(* CoDeSys 2.3.9.52 project: dom1.pro *)
(* Libraries: Standard.lib 8.11.10 11:37:48, SYSLIBCALLBACK.LIB 8.11.10 11:37:48 *)

(* PLC configuration (modules and I/O channels)
0750-0430 8 DI 24 V DC 3.0ms [Type_1_8_Channels] node 0, in %IB0 out %QB0 {INTTypePAAssignment = PLC; INTTypeModule = plugged}
  AT %IX0.0 [BOOLOnX_I] Ch_1 Digital input
  AT %IX0.1 [BOOLOnX_I] Ch_2 Digital input
  AT %IX0.2 [BOOLOnX_I] Ch_3 Digital input
  AT %IX0.3 [BOOLOnX_I] Ch_4 Digital input
  AT %IX0.4 [BOOLOnX_I] Ch_5 Digital input
  AT %IX0.5 [BOOLOnX_I] Ch_6 Digital input
  AT %IX0.6 [BOOLOnX_I] Ch_7 Digital input
  AT %IX0.7 [BOOLOnX_I] Ch_8 Digital input
0750-0430 8 DI 24 V DC 3.0ms [Type_1_8_Channels] node 1, in %IB0 out %QB0 {INTTypePAAssignment = PLC; INTTypeModule = plugged}
  AT %IX0.8 [BOOLOnX_I] Ch_1 Digital input
  AT %IX0.9 [BOOLOnX_I] Ch_2 Digital input
  AT %IX0.10 [BOOLOnX_I] Ch_3 Digital input
  AT %IX0.11 [BOOLOnX_I] Ch_4 Digital input
  AT %IX0.12 [BOOLOnX_I] Ch_5 Digital input
  AT %IX0.13 [BOOLOnX_I] Ch_6 Digital input
  AT %IX0.14 [BOOLOnX_I] Ch_7 Digital input
  AT %IX0.15 [BOOLOnX_I] Ch_8 Digital input
0750-0430 8 DI 24 V DC 3.0ms [Type_1_8_Channels] node 2, in %IB1 out %QB0 {INTTypePAAssignment = PLC; INTTypeModule = plugged}
  AT %IX1.0 [BOOLOnX_I] Ch_1 Digital input
  AT %IX1.1 [BOOLOnX_I] Ch_2 Digital input
  AT %IX1.2 [BOOLOnX_I] Ch_3 Digital input
  AT %IX1.3 [BOOLOnX_I] Ch_4 Digital input
  AT %IX1.4 [BOOLOnX_I] Ch_5 Digital input
  AT %IX1.5 [BOOLOnX_I] Ch_6 Digital input
  AT %IX1.6 [BOOLOnX_I] Ch_7 Digital input
  AT %IX1.7 [BOOLOnX_I] Ch_8 Digital input
0750-0430 8 DI 24 V DC 3.0ms [Type_1_8_Channels] node 3, in %IB2 out %QB0 {INTTypePAAssignment = PLC; INTTypeModule = plugged}
  AT %IX1.8 [BOOLOnX_I] Ch_1 Digital input
  AT %IX1.9 [BOOLOnX_I] Ch_2 Digital input
  AT %IX1.10 [BOOLOnX_I] Ch_3 Digital input
  AT %IX1.11 [BOOLOnX_I] Ch_4 Digital input
  AT %IX1.12 [BOOLOnX_I] Ch_5 Digital input
  AT %IX1.13 [BOOLOnX_I] Ch_6 Digital input
  AT %IX1.14 [BOOLOnX_I] Ch_7 Digital input
  AT %IX1.15 [BOOLOnX_I] Ch_8 Digital input
0750-0430 8 DI 24 V DC 3.0ms [Type_1_8_Channels] node 4, in %IB3 out %QB0 {INTTypePAAssignment = PLC; INTTypeModule = plugged}
  AT %IX2.0 [BOOLOnX_I] Ch_1 Digital input
  AT %IX2.1 [BOOLOnX_I] Ch_2 Digital input
  AT %IX2.2 [BOOLOnX_I] Ch_3 Digital input
  AT %IX2.3 [BOOLOnX_I] Ch_4 Digital input
  AT %IX2.4 [BOOLOnX_I] Ch_5 Digital input
  AT %IX2.5 [BOOLOnX_I] Ch_6 Digital input
  AT %IX2.6 [BOOLOnX_I] Ch_7 Digital input
  AT %IX2.7 [BOOLOnX_I] Ch_8 Digital input
0750-0430 8 DI 24 V DC 3.0ms [Type_1_8_Channels] node 5, in %IB4 out %QB0 {INTTypePAAssignment = PLC; INTTypeModule = plugged}
  AT %IX2.8 [BOOLOnX_I] Ch_1 Digital input
  AT %IX2.9 [BOOLOnX_I] Ch_2 Digital input
  AT %IX2.10 [BOOLOnX_I] Ch_3 Digital input
  AT %IX2.11 [BOOLOnX_I] Ch_4 Digital input
  AT %IX2.12 [BOOLOnX_I] Ch_5 Digital input
  AT %IX2.13 [BOOLOnX_I] Ch_6 Digital input
  AT %IX2.14 [BOOLOnX_I] Ch_7 Digital input
  AT %IX2.15 [BOOLOnX_I] Ch_8 Digital input
0750-0430 8 DI 24 V DC 3.0ms [Type_1_8_Channels] node 6, in %IB5 out %QB0 {INTTypePAAssignment = PLC; INTTypeModule = plugged}
  AT %IX3.0 [BOOLOnX_I] Ch_1 Digital input
  AT %IX3.1 [BOOLOnX_I] Ch_2 Digital input
  AT %IX3.2 [BOOLOnX_I] Ch_3 Digital input
  AT %IX3.3 [BOOLOnX_I] Ch_4 Digital input
  AT %IX3.4 [BOOLOnX_I] Ch_5 Digital input
  AT %IX3.5 [BOOLOnX_I] Ch_6 Digital input
  AT %IX3.6 [BOOLOnX_I] Ch_7 Digital input
  AT %IX3.7 [BOOLOnX_I] Ch_8 Digital input
0750-0430 8 DI 24 V DC 3.0ms [Type_1_8_Channels] node 7, in %IB6 out %QB0 {INTTypePAAssignment = PLC; INTTypeModule = plugged}
  AT %IX3.8 [BOOLOnX_I] Ch_1 Digital input
  AT %IX3.9 [BOOLOnX_I] Ch_2 Digital input
  AT %IX3.10 [BOOLOnX_I] Ch_3 Digital input
  AT %IX3.11 [BOOLOnX_I] Ch_4 Digital input
  AT %IX3.12 [BOOLOnX_I] Ch_5 Digital input
  AT %IX3.13 [BOOLOnX_I] Ch_6 Digital input
  AT %IX3.14 [BOOLOnX_I] Ch_7 Digital input
  AT %IX3.15 [BOOLOnX_I] Ch_8 Digital input
0750-0430 8 DI 24 V DC 3.0ms [Type_1_8_Channels] node 8, in %IB7 out %QB0 {INTTypePAAssignment = PLC; INTTypeModule = plugged}
  AT %IX4.0 [BOOLOnX_I] Ch_1 Digital input
  AT %IX4.1 [BOOLOnX_I] Ch_2 Digital input
  AT %IX4.2 [BOOLOnX_I] Ch_3 Digital input
  AT %IX4.3 [BOOLOnX_I] Ch_4 Digital input
  AT %IX4.4 [BOOLOnX_I] Ch_5 Digital input
  AT %IX4.5 [BOOLOnX_I] Ch_6 Digital input
  AT %IX4.6 [BOOLOnX_I] Ch_7 Digital input
  AT %IX4.7 [BOOLOnX_I] Ch_8 Digital input
0750-0430 8 DI 24 V DC 3.0ms [Type_1_8_Channels] node 9, in %IB8 out %QB0 {INTTypePAAssignment = PLC; INTTypeModule = plugged}
  AT %IX4.8 [BOOLOnX_I] Ch_1 Digital input
  AT %IX4.9 [BOOLOnX_I] Ch_2 Digital input
  AT %IX4.10 [BOOLOnX_I] Ch_3 Digital input
  AT %IX4.11 [BOOLOnX_I] Ch_4 Digital input
  AT %IX4.12 [BOOLOnX_I] Ch_5 Digital input
  AT %IX4.13 [BOOLOnX_I] Ch_6 Digital input
  AT %IX4.14 [BOOLOnX_I] Ch_7 Digital input
  AT %IX4.15 [BOOLOnX_I] Ch_8 Digital input
0750-0530 8 DO 24 V DC 0.5A [Type_10_8_Channels] node 10, in %IB9 out %QB0 {INTTypePAAssignment = PLC; INTTypeModule = plugged}
  K1_2a AT %QX0.0 [BOOLOnX_Q] Ch_1 Digital output
  K1_2b AT %QX0.1 [BOOLOnX_Q] Ch_2 Digital output
  L1_1a AT %QX0.2 [BOOLOnX_Q] Ch_3 Digital output
  L1_1b AT %QX0.3 [BOOLOnX_Q] Ch_4 Digital output
  N1_1a AT %QX0.4 [BOOLOnX_Q] Ch_5 Digital output
  N1_1b AT %QX0.5 [BOOLOnX_Q] Ch_6 Digital output
  E2_1a AT %QX0.6 [BOOLOnX_Q] Ch_7 Digital output
  E2_1b AT %QX0.7 [BOOLOnX_Q] Ch_8 Digital output
0750-0530 8 DO 24 V DC 0.5A [Type_10_8_Channels] node 11, in %IB10 out %QB0 {INTTypePAAssignment = PLC; INTTypeModule = plugged}
  S2_1a AT %QX0.8 [BOOLOnX_Q] Ch_1 Digital output
  S2_1b AT %QX0.9 [BOOLOnX_Q] Ch_2 Digital output
  S3_1a AT %QX0.10 [BOOLOnX_Q] Ch_3 Digital output
  S3_1b AT %QX0.11 [BOOLOnX_Q] Ch_4 Digital output
  S4_3a AT %QX0.12 [BOOLOnX_Q] Ch_5 Digital output
  S4_3b AT %QX0.13 [BOOLOnX_Q] Ch_6 Digital output
  Z7_1a AT %QX0.14 [BOOLOnX_Q] Ch_7 Digital output
  Z7_1b AT %QX0.15 [BOOLOnX_Q] Ch_8 Digital output
0750-0530 8 DO 24 V DC 0.5A [Type_10_8_Channels] node 12, in %IB10 out %QB1 {INTTypePAAssignment = PLC; INTTypeModule = plugged}
  J5_1a AT %QX1.0 [BOOLOnX_Q] Ch_1 Digital output
  J5_1b AT %QX1.1 [BOOLOnX_Q] Ch_2 Digital output
  A1_2 AT %QX1.2 [BOOLOnX_Q] Ch_3 Digital output
  H1_1 AT %QX1.3 [BOOLOnX_Q] Ch_4 Digital output
  H6_1 AT %QX1.4 [BOOLOnX_Q] Ch_5 Digital output
  H7_1 AT %QX1.5 [BOOLOnX_Q] Ch_6 Digital output
  P1_1 AT %QX1.6 [BOOLOnX_Q] Ch_7 Digital output
  P3_1 AT %QX1.7 [BOOLOnX_Q] Ch_8 Digital output
0750-0530 8 DO 24 V DC 0.5A [Type_10_8_Channels] node 13, in %IB10 out %QB2 {INTTypePAAssignment = PLC; INTTypeModule = plugged}
  P5_1 AT %QX1.8 [BOOLOnX_Q] Ch_1 Digital output
  K11_1 AT %QX1.9 [BOOLOnX_Q] Ch_2 Digital output
  S15_1a AT %QX1.10 [BOOLOnX_Q] Ch_3 Digital output
  S15_1b AT %QX1.11 [BOOLOnX_Q] Ch_4 Digital output
  N7_1 AT %QX1.12 [BOOLOnX_Q] Ch_5 Digital output
  L5_1 AT %QX1.13 [BOOLOnX_Q] Ch_6 Digital output
  L4_1 AT %QX1.14 [BOOLOnX_Q] Ch_7 Digital output
  E6_1 AT %QX1.15 [BOOLOnX_Q] Ch_8 Digital output
0750-0530 8 DO 24 V DC 0.5A [Type_10_8_Channels] node 14, in %IB10 out %QB3 {INTTypePAAssignment = PLC; INTTypeModule = plugged}
  S14_1a AT %QX2.0 [BOOLOnX_Q] Ch_1 Digital output
  S14_1b AT %QX2.1 [BOOLOnX_Q] Ch_2 Digital output
  S16_1a AT %QX2.2 [BOOLOnX_Q] Ch_3 Digital output
  S16_1b AT %QX2.3 [BOOLOnX_Q] Ch_4 Digital output
  S25_1 AT %QX2.4 [BOOLOnX_Q] Ch_5 Digital output
  S26_2 AT %QX2.5 [BOOLOnX_Q] Ch_6 Digital output
  S28_1a AT %QX2.6 [BOOLOnX_Q] Ch_7 Digital output
  S28_1b AT %QX2.7 [BOOLOnX_Q] Ch_8 Digital output
  G3_1 AT %QX2.8 [BOOLOnX_Q] Ch_1 Digital output
  J2_1 AT %QX2.9 [BOOLOnX_Q] Ch_2 Digital output
  B1_1 AT %QX2.10 [BOOLOnX_Q] Ch_3 Digital output
  B2_2 AT %QX2.11 [BOOLOnX_Q] Ch_4 Digital output
  Z1_1a AT %QX2.12 [BOOLOnX_Q] Ch_5 Digital output
  S12_1 AT %QX2.13 [BOOLOnX_Q] Ch_6 Digital output
  W1_1 AT %QX2.14 [BOOLOnX_Q] Ch_7 Digital output
  AT %QX2.15 [BOOLOnX_Q] Ch_8 Digital output
  AT %QX3.0 [BOOLOnX_Q] Ch_1 Digital output
  AT %QX3.1 [BOOLOnX_Q] Ch_2 Digital output
  AT %QX3.2 [BOOLOnX_Q] Ch_3 Digital output
  AT %QX3.3 [BOOLOnX_Q] Ch_4 Digital output
  AT %QX3.4 [BOOLOnX_Q] Ch_5 Digital output
  AT %QX3.5 [BOOLOnX_Q] Ch_6 Digital output
  AT %QX3.6 [BOOLOnX_Q] Ch_7 Digital output
  AT %QX3.7 [BOOLOnX_Q] Ch_8 Digital output
Fieldbus variables [FB_VARS] node 1, in %IB0 out %QB0
Flag variables [FLAG_VARS] node 2, in %IB0 out %QB0
Modbus-Master [MB_MASTER] node 3, in %IB0 out %QB0
*)

(* Task configuration *)
TASK clock1s (PRIORITY := 3, INTERVAL := T#1000ms);
	clock1s();
END_TASK
TASK loop (PRIORITY := 2);
	PLC_PRG();
	V2();
END_TASK
TASK clock01s (PRIORITY := 1, INTERVAL := T#100ms);
	clock01s()
END_TASK

(* Global variable list: Global_Variables *)
VAR_GLOBAL
	clock1secImpulse:BOOL;
	clock01secImpulse:BOOL;

	testA AT %MB0:INT;


	B3_3a AT %IX0.0:BOOL;
	B3_3b AT %IX0.1:BOOL;
	E5_1a AT %IX0.2:BOOL;
	E5_1b AT %IX0.3:BOOL;
	H3_1a AT %IX0.4:BOOL;
	H3_1b AT %IX0.5:BOOL;
	H5_1a AT %IX0.6:BOOL;
	H5_1b AT %IX0.7:BOOL;
	H5_1c AT %IX0.8:BOOL;
	H5_1d AT %IX0.9:BOOL;
	H11_1a AT %IX0.10:BOOL;
	H11_1b AT %IX0.11:BOOL;
	J8_1a AT %IX0.12:BOOL;
	J8_1b AT %IX0.13:BOOL;
	J8_1c AT %IX0.14:BOOL;
	K5_2a AT %IX0.15:BOOL;
	K5_2b AT %IX1.0:BOOL;
	K5_3a AT %IX1.1:BOOL;
	K5_3b AT %IX1.2:BOOL;
	L4_3a AT %IX1.3:BOOL;
	L4_3b AT %IX1.4:BOOL;
	L4_3c AT %IX1.5:BOOL;
	L4_3d AT %IX1.6:BOOL;
	P7_1a AT %IX1.7:BOOL;
	P7_1b AT %IX1.8:BOOL;
	P8_1a AT %IX1.9:BOOL;
	P8_1b AT %IX1.10:BOOL;
	P9_1a AT %IX1.11:BOOL;
	P9_1b AT %IX1.12:BOOL;
	S1_2a AT %IX1.13:BOOL;
	S1_2b AT %IX1.14:BOOL;
	S1_2c AT %IX1.15:BOOL;
	S1_2d AT %IX2.0:BOOL;
	S1_2e AT %IX2.1:BOOL;
	S1_2f AT %IX2.2:BOOL;
	S2_2a AT %IX2.3:BOOL;
	S2_2b AT %IX2.4:BOOL;
	S3_4a AT %IX2.5:BOOL;
	S3_4b AT %IX2.6:BOOL;
	S4_1a AT %IX2.7:BOOL;
	S4_1b AT %IX2.8:BOOL;
	S4_1c AT %IX2.9:BOOL;
	S4_1d AT %IX2.10:BOOL;
	S4_1e AT %IX2.11:BOOL;
	S4_1f AT %IX2.12:BOOL;
	S24_1a AT %IX2.13:BOOL;
	S24_1b AT %IX2.14:BOOL;
	S27_1a AT %IX2.15:BOOL;
	S27_1b AT %IX3.0:BOOL;
	W2_1a AT %IX3.1:BOOL;
	Z12_1a AT %IX3.2:BOOL;
	Z12_1b AT %IX3.3:BOOL;
	Z12_1c AT %IX3.4:BOOL;
	N6_1a AT %IX3.5:BOOL;
	N6_1b AT %IX3.6:BOOL;
	H9_2a AT %IX3.7:BOOL;
	H9_2b AT %IX3.8:BOOL;
	H9_2c AT %IX3.9:BOOL;
	H9_2d AT %IX3.10:BOOL;
	E2_3a AT %IX3.11:BOOL;
	E2_3b AT %IX3.12:BOOL;
	K1_1a AT %IX3.13:BOOL;
	K1_1b AT %IX3.14:BOOL;
	J10_2a AT %IX3.15:BOOL;
	J10_2b AT %IX4.0:BOOL;
	N1_2a AT %IX4.1:BOOL;
	N1_2b AT %IX4.2:BOOL;
	Z11_1a AT %IX4.3:BOOL;
	Z11_1b AT %IX4.4:BOOL;

	K3_3 AT %QX2.15:BOOL;
	Z3_1a AT %QX3.0:BOOL;
	Z3_1b AT %QX3.1:BOOL;
	Z4_1a AT %QX3.2:BOOL;
	Z4_1b AT %QX3.3:BOOL;
	J1_1a AT %QX3.4:BOOL;
	J1_1b AT %QX3.5:BOOL;
	P2_1a AT %QX3.6:BOOL;
	P2_1b AT %QX3.7:BOOL;

	lastInput AT%IX4.15:BOOL;
END_VAR

(* Global variable list: Shaders *)
VAR_GLOBAL
	shader_kuchnia:Shader;
	shader_taras:Shader;
	shader_kominek:Shader;
	shader_gabinet:Shader;
	shader_sypialnia:Shader;
	shader_lazienka:Shader;
	shader_kotlownia:Shader;
	shader_Julka:Shader;
	shader_Julka_dach:Shader;
	shader_Zosia:Shader;
	shader_Zosia_dach_L:Shader;
	shader_Zosia_dach_P:Shader;
	shader_przedpokoj:Shader;

END_VAR

(* POU clock1s, ST *)
PROGRAM clock1s
VAR
END_VAR
clock1secImpulse:=1;
END_PROGRAM

(* POU PLC_PRG, ST *)
PROGRAM PLC_PRG
VAR
	firstLoop:BOOL;
	test:INT;

	Attic:Attic;
	Bathroom_pietro:Bathroom_pietro;
	E_gabinet:E_gabinet;
	Garderoba:Garderoba;
	Hol_parter:Hol_parter;
	Julka:Julka;
	Kotlownia:Kotlownia;
	Lazienka_parter:Lazienka_parter;
	N_sypialnia:N_sypialnia;
	Przedpokoj_pietro:Przedpokoj_pietro;
	Salon:Salon;
	Zosia:Zosia;
	Taras:Taras;

	LockMode:LockMode;

END_VAR
IF NOT firstLoop THEN
	firstLoop:=1;
	start();
END_IF

lockMode();

attic();
bathroom_pietro();
e_gabinet();
garderoba();
hol_parter();
julka();
kotlownia(presenceDetection:=bathroom_pietro.presenceDetection XOR lazienka_parter.presenceDetection XOR salon.kuchniaPresenceDetection );
lazienka_parter();
n_sypialnia();
przedpokoj_pietro();
salon();
zosia();
taras();

clock1secImpulse := 0;
clock01secImpulse:=0;
test := test + 1;
END_PROGRAM

(* POU Rooms/Attic, ST *)
FUNCTION_BLOCK Attic
VAR
	lamps:ButtonTriggeredTimedOnOff:= (timeSetup:= 400);
END_VAR
lamps(input:=P7_1b, output => A1_2);
END_FUNCTION_BLOCK

(* POU Components/OnOff/ButtonTriggeredTimedOnOff, ST *)
FUNCTION_BLOCK ButtonTriggeredTimedOnOff
VAR_INPUT
	input:BOOL;
	timeSetup:INT;
END_VAR
VAR_OUTPUT
	output:BOOL;
END_VAR
VAR
	Button:Button;
	TimedOnOff:TimedOnOff;
	state:BOOL;
END_VAR
button(input:=input);
timedOnOff(timeSetup:=timeSetup, input:= button.fallingEdge, permanent:= button.longPressed, output=>output);
state:=timedOnOff.state;
END_FUNCTION_BLOCK

(* POU Components/Button, ST *)
FUNCTION_BLOCK Button
VAR_INPUT
	input: BOOL;
END_VAR

VAR
	EdgeDetection:EdgeDetection := (onFallingEdge:=1);
	fallingEdge:BOOL;
	longPressed:BOOL;
	timer:Delay:= (timeSetup:= 10);
	tmp:BOOL;
END_VAR
EdgeDetection(input:=input, output => tmp);
fallingEdge := tmp AND NOT timer.afterTime;

timer(start:= input);
longPressed:= timer.afterTimeImpulse;
END_FUNCTION_BLOCK

(* POU Components/EdgeDetection, ST *)
FUNCTION_BLOCK EdgeDetection
VAR_INPUT
	input:BOOL;
	onFallingEdge:BOOL;
	onRisingEdge:BOOL;
END_VAR
VAR_OUTPUT
	output: BOOL;
END_VAR
VAR
	oldValue: BOOL;
	impulse:BOOL;
END_VAR
VAR_IN_OUT
END_VAR
output:= (oldValue XOR input) AND ((onFallingEdge AND oldValue) OR (onRisingEdge AND NOT oldValue));
impulse:=output;
oldValue:= input;
END_FUNCTION_BLOCK

(* POU Components/Delay, ST *)
FUNCTION_BLOCK Delay
VAR_INPUT
	start:BOOL;
	stop:BOOL;
	timeSetup: INT;  (*  x0.1sec  *)
	resetTime:BOOL;
END_VAR
VAR_OUTPUT
END_VAR
VAR
	afterTime:BOOL;
	afterTimeImpulse:BOOL;
	untilTimePass:BOOL;
	counter: INT;
END_VAR
IF NOT start  OR stop OR resetTime THEN
	counter := 0;
END_IF

IF clock01secImpulse AND start THEN
	counter := counter + 1;
END_IF
IF counter > timeSetup THEN
	counter := timeSetup;
END_IF

afterTimeImpulse:= NOT afterTime AND counter >= timeSetup;
afterTime := counter >= timeSetup;

untilTimePass := start AND (NOT stop) AND counter < timeSetup;
END_FUNCTION_BLOCK

(* POU start, ST *)
PROGRAM start
VAR

	test0 AT %QX0.0:BOOL;
END_VAR
test0 := 0;
END_PROGRAM

(* POU Components/OnOff/TimedOnOff, ST *)
FUNCTION_BLOCK TimedOnOff
VAR_INPUT
	permanent:BOOL;
	input:BOOL;
	postpone:BOOL;
	timeSetup:INT;
	state:BOOL;
END_VAR
VAR_OUTPUT
	output:BOOL;
END_VAR
VAR
	timer:Delay;
	permanentMode: BOOL;
END_VAR
timer.timeSetup:=timeSetup;

IF input THEN
	state:= NOT state;
END_IF

IF permanent THEN
	permanentMode:=1;
	state:=1;
END_IF

IF NOT state THEN
	permanentMode:= 0;
END_IF;

timer.resetTime:=postpone;
IF postpone THEN
	state:=1;
END_IF

timer(start:=state);

IF timer.afterTimeImpulse AND NOT permanentMode THEN
	state := 0;
END_IF

output:=state;
END_FUNCTION_BLOCK

(* POU Rooms/Bathroom_pietro, ST *)
FUNCTION_BLOCK  Bathroom_pietro
VAR
	mainLamp:OnOff;
	wallLamp:OnOff;
	presenceDetection:BOOL;
END_VAR
mainLamp(input:=B3_3a OR P9_1a, output => B1_1);
wallLamp(input:=B3_3b, output => B2_2);

presenceDetection:=B3_3a XOR B3_3b XOR P9_1a XOR P9_1b;
END_FUNCTION_BLOCK

(* POU Components/OnOff/OnOff, ST *)
FUNCTION_BLOCK OnOff

VAR_INPUT
	input:BOOL;
	state:BOOL;
END_VAR

VAR_OUTPUT
	output:BOOL;
END_VAR

VAR
	EdgeDetection:EdgeDetection := (onFallingEdge:=1);
	tmp:BOOL;
END_VAR
EdgeDetection(input:=input, output => tmp);

IF tmp THEN
	state := NOT state;
END_IF

output := state;
END_FUNCTION_BLOCK

(* POU Rooms/E_gabinet, ST *)
FUNCTION_BLOCK E_gabinet
VAR
	mainLamp:OnOff;
	Shader: ButtonTriggeredShader;
END_VAR
mainLamp(input:=E5_1b, output => E6_1);

shader(input:=E5_1a, shader:=shader_gabinet, openOut=>E2_1a, closeOut=>E2_1b);
END_FUNCTION_BLOCK

(* POU Components/Shader/Shader, ST *)
FUNCTION_BLOCK Shader
VAR_INPUT
(*	open:BOOL;
	close:BOOL;*)
	openImpulse:BOOL;
	closeImpulse:BOOL;
	switch:BOOL;
END_VAR
VAR
	closing: BOOL;
	opening: BOOL;
	lastDirection:BOOL;
	delayTimer:Delay := (timeSetup:= 400);
	state:INT;  (* 0: closed; 100: open *)
END_VAR
delayTimer();

IF delayTimer.afterTime OR ( (openImpulse OR closeImpulse OR switch) AND (closing OR opening) ) THEN
	delayTimer.start := 0;
	closing := 0;
	opening := 0;
ELSE
	IF switch THEN
		lastDirection:= NOT lastDirection;
		closing:=lastDirection;
		opening:=NOT lastDirection;
		delayTimer.start := 1;
	END_IF

	IF openImpulse AND NOT closing THEN
		lastDirection:=0;
		closing := 0;
		opening := 1;
		delayTimer.start := 1;
	END_IF

	IF closeImpulse AND NOT opening THEN
		lastDirection:=1;
		closing := 1;
		opening := 0;
		delayTimer.start := 1;
	END_IF
END_IF

openImpulse:=0;
closeImpulse:=0;
END_FUNCTION_BLOCK

(* POU Components/Shader/ButtonTriggeredShader, ST *)
FUNCTION_BLOCK ButtonTriggeredShader
VAR_INPUT
	input:BOOL;
END_VAR
VAR_OUTPUT
	closeOut:BOOL;
	openOut:BOOL;
END_VAR
VAR
	Button:Button;
END_VAR
VAR_IN_OUT
	Shader:Shader;
END_VAR
button(input:=input);
shader(switch:= button.fallingEdge);

closeOut:= shader.closing;
openOut:= shader.opening;
END_FUNCTION_BLOCK

(* POU Rooms/Garderoba, ST *)
FUNCTION_BLOCK Garderoba
VAR
	mainLamp:ButtonTriggeredTimedOnOff:= (timeSetup:= 12000);
END_VAR
mainLamp(input:=H3_1b, output => G3_1);
END_FUNCTION_BLOCK

(* POU Rooms/Hol_parter, ST *)
FUNCTION_BLOCK Hol_parter
VAR
(*	lampNextToL:OnOff; *)
	lampNextToL:ButtonTriggeredTimedOnOff:= (timeSetup:= 200);
	mainLamp:ButtonTriggeredTimedOnOff:= (timeSetup:= 6000);
	entranceLamp:ButtonTriggeredTimedOnOff:= (timeSetup:= 1200);

	tmp: BOOL;
END_VAR
mainLamp(input:=H9_2a OR S1_2d, output => H7_1);

lampNextToL(input:=H9_2b OR H3_1a);
H1_1:= lampNextToL.state;
H6_1:=lampNextToL.state;

entranceLamp(input:=H9_2c AND NOT H9_2d, output => W1_1);
END_FUNCTION_BLOCK

(* POU Rooms/Julka, ST *)
FUNCTION_BLOCK Julka
VAR
	mainLamp :OnOff;
(*	buttonJ8_1b: Button;
	shaderJ:Shader;
*)
	Shader: ButtonTriggeredShader;
	shader_dach: ButtonTriggeredShader;
END_VAR
mainLamp(input:=J8_1c, output => J2_1);

shader(input:=J8_1b, shader:=shader_Julka, openOut=>J5_1a, closeOut=>J5_1b);
shader_dach(input:=J8_1a, shader:=shader_Julka_dach, openOut=>J1_1a, closeOut=>J1_1b);

(*
buttonJ8_1b(input:=J8_1b);
shaderJ(switch:=buttonJ8_1b.fallingEdge);
J5_1a:=shaderJ.opening;
J5_1b:=shaderJ.closing;*)
END_FUNCTION_BLOCK

(* POU Rooms/Kotlownia, ST *)
FUNCTION_BLOCK Kotlownia
VAR_INPUT
	presenceDetection:BOOL;
END_VAR
VAR
	mainLamp:ButtonTriggeredTimedOnOff:= (timeSetup:= 12000);
	Shader:ButtonTriggeredShader;

	hotWaterDemandTimer:Delay:= (timeSetup:= 18000);
	EdgeDetection:EdgeDetection := (onRisingEdge:=1, onFallingEdge:=1);
	startPumpImpulse:BOOL;
	circulatingPumpPWM:PWMTimer:= (onTimeSetup:= 600, offTimeSetup:=18000);
END_VAR
mainLamp(input:=K5_3a OR K5_2b, output => K11_1);
shader(input:=K5_3b OR K5_2a, shader:=shader_kotlownia, openOut=>K1_2a, closeOut=>K1_2b);

edgeDetection(input:=presenceDetection);
hotWaterDemandTimer(start:=1, resetTime:=edgeDetection.impulse);
circulatingPumpPWM(start:=hotWaterDemandTimer.untilTimePass, output => K3_3);
END_FUNCTION_BLOCK

(* POU Components/OnOff/PWMTimer, ST *)
FUNCTION_BLOCK PWMTimer
VAR_INPUT
	start:BOOL;
	onTimeSetup:INT;
	offTimeSetup:INT;
END_VAR
VAR_OUTPUT
	output:BOOL;
END_VAR
VAR
	onTimer:Delay;
	offTimer:Delay;
END_VAR
onTimer.timeSetup:=onTimeSetup;
offTimer.timeSetup:=offTimeSetup;

onTimer(start:=start);
offTimer(start:=onTimer.afterTime);
onTimer.resetTime:=offTimer.afterTimeImpulse;
output:= onTimer.untilTimePass;
END_FUNCTION_BLOCK

(* POU Rooms/Lazienka_parter, ST *)
FUNCTION_BLOCK Lazienka_parter
VAR
	mainLamp:OnOff;
	wallLamp:OnOff;
	Shader: ButtonTriggeredShader;
	presenceDetection:BOOL;
END_VAR
mainLamp(input:=H5_1a OR L4_3a, output => L5_1);
wallLamp(input:=H5_1b OR L4_3b, output => L4_1);

shader(input:=H5_1c OR L4_3c, shader:=shader_lazienka, openOut=>L1_1a, closeOut=>L1_1b);

presenceDetection:=H5_1a XOR H5_1b XOR H5_1c XOR H5_1d XOR L4_3a XOR L4_3b XOR L4_3c XOR L4_3d;
END_FUNCTION_BLOCK

(* POU Rooms/N_sypialnia, ST *)
FUNCTION_BLOCK N_sypialnia
VAR
	mainLamp:OnOff;
	Shader: ButtonTriggeredShader;
END_VAR
mainLamp(input:=N6_1b, output => N7_1);
shader(input:=N6_1a, shader:=shader_sypialnia, openOut=>N1_1a, closeOut=>N1_1b);
END_FUNCTION_BLOCK

(* POU Rooms/Przedpokoj_pietro, ST *)
FUNCTION_BLOCK Przedpokoj_pietro
VAR
	mainLamp:ButtonTriggeredTimedOnOff:= (timeSetup:= 300);
	Shader: ButtonTriggeredShader;
	tmp: BOOL;
END_VAR
mainLamp(input:=H11_1a OR P7_1a OR P8_1a);
P1_1:= mainLamp.state;
P3_1:=mainLamp.state;

shader(input:=H11_1b, shader:=shader_przedpokoj, openOut=>P2_1a, closeOut=>P2_1b);
END_FUNCTION_BLOCK

(* POU Rooms/Salon, ST *)
FUNCTION_BLOCK Salon
VAR
	kuchniaS:Scene := (count:=4);
	kuchnia:ButtonTriggeredScene;

	wyspaS:Scene := (count:=4);
	wyspa:ButtonTriggeredScene;

	kominekS:Scene := (count:=4);
	kominek:ButtonTriggeredScene;

	ledLeft:OnOff;
	ledRight:OnOff;
	jadalnia:OnOff;

	kuchniaMain:SceneGroup;

	kuchniaShader: ButtonTriggeredShader;
	tarasShader: ButtonTriggeredShader;
	kominekShader: ButtonTriggeredShader;

	kuchniaPresenceDetection:BOOL;
END_VAR
(*
S1.2 przy wejsciu
S2.2 przy kominku
S3.4 prawo od okna
S4.1 przy tarasie
S24.1 blat po prawej
S27.1 blat po lewej
*)
kuchniaMain(switch:=S1_2a OR S4_1c, a:=kuchniaS.enabled, b:=wyspaS.enabled, c:=ledLeft.state, d:=ledRight.state);
kuchnia(input:=S3_4b OR S24_1a, scene:=kuchniaS, a=> S16_1a, b=>S16_1b);
wyspa(input:=S4_1e OR S27_1a OR S1_2e, scene:=wyspaS,  a=> S28_1a, b=>S28_1b);
ledLeft(input:=S27_1b, output => S26_2);
ledRight(input:=S24_1b, output => S25_1);
jadalnia(input:=S4_1b OR S1_2b, output => S15_1b);
kominek(input:=S1_2c OR S2_2a, scene:=kominekS, a=> S14_1a, b=>S14_1b);

kuchniaShader(input:=S3_4a, shader:=shader_kuchnia, openOut=>S3_1a, closeOut=>S3_1b);
tarasShader(input:=S4_1a, shader:=shader_taras, openOut=>S4_3a, closeOut=>S4_3b);
kominekShader(input:=S2_2b, shader:=shader_kominek, openOut=>S2_1a, closeOut=>S2_1b);

kuchniaPresenceDetection:=S1_2a XOR S4_1c XOR S24_1a XOR S24_1b XOR S27_1a XOR S27_1b XOR S3_4a XOR S3_4b;
END_FUNCTION_BLOCK

(* POU Components/Scene/Scene, ST *)
FUNCTION_BLOCK Scene
VAR_INPUT
	rotate:BOOL;
	switch:BOOL;
END_VAR

VAR
	count:INT:=3;
	number:INT;
	enabled:BOOL;
	privateNumber:INT;
END_VAR
enabled:= enabled XOR switch;

IF rotate AND enabled THEN
	privateNumber := privateNumber + 1;
END_IF

IF privateNumber >= count OR privateNumber < 1 THEN
	privateNumber:=1;
END_IF

IF enabled THEN
	number := privateNumber;
ELSE
	number := 0;
END_IF
END_FUNCTION_BLOCK

(* POU Components/Scene/ButtonTriggeredScene, ST *)
FUNCTION_BLOCK ButtonTriggeredScene
VAR_INPUT
	input:BOOL;
END_VAR
VAR_OUTPUT
	a:BOOL;
	b:BOOL;
END_VAR
VAR
	Button:Button;
END_VAR
VAR_IN_OUT
	Scene:Scene;
END_VAR
button(input:=input);
scene(rotate:= button.longPressed, switch:= button.fallingEdge);
a:= scene.number = 1 OR scene.number = 2;
b:= scene.number = 1 OR scene.number = 3;
END_FUNCTION_BLOCK

(* POU Components/Scene/SceneGroup, ST *)
FUNCTION_BLOCK SceneGroup
VAR_INPUT
	switch:BOOL;
END_VAR
VAR_OUTPUT
END_VAR
VAR
	lastState: ARRAY [0..3] OF BOOL;
	Button:Button;

	tmp1:BOOL;
END_VAR
VAR_IN_OUT
	a:BOOL;
	b:BOOL;
	c:BOOL;
	d:BOOL;
END_VAR
button(input:=switch);
IF button.fallingEdge THEN
	IF a OR b OR c OR d THEN
		lastState[0]:=a;
		lastState[1]:=b;
		lastState[2]:=c;
		lastState[3]:=d;
		a:=0;
		b:=0;
		c:=0;
		d:=0;
	ELSE
		a:=lastState[0];
		b:=lastState[1];
		c:=lastState[2];
		d:=lastState[3];
	END_IF
END_IF
END_FUNCTION_BLOCK

(* POU Rooms/Zosia, ST *)
FUNCTION_BLOCK Zosia
VAR
	mainLamp: OnOff;
(*	buttonZ12_1b: Button;*)
	Shader: ButtonTriggeredShader;
	shader_dach_L: ButtonTriggeredShader;
	shader_dach_P: ButtonTriggeredShader;
(*	shaderZ:Shader;*)
END_VAR
mainLamp(input:=Z12_1a, output => Z1_1a);

shader(input:=Z12_1b, shader:=shader_Zosia, openOut=>Z7_1a, closeOut=>Z7_1b);
shader_dach_L(input:=Z12_1c, shader:=shader_Zosia_dach_L, openOut=>Z3_1a, closeOut=>Z3_1b);
shader_dach_P(input:=Z12_1c, shader:=shader_Zosia_dach_P, openOut=>Z4_1a, closeOut=>Z4_1b);

(*
buttonZ12_1b(input:=Z12_1b);
shaderZ(switch:=buttonZ12_1b.fallingEdge);
Z7_1a:=shaderZ.opening;
Z7_1b:=shaderZ.closingc
*)
END_FUNCTION_BLOCK

(* POU Rooms/Taras, ST *)
FUNCTION_BLOCK Taras
VAR_INPUT
END_VAR
VAR_OUTPUT
END_VAR
VAR
	mainLamp:ButtonTriggeredTimedOnOff:= (timeSetup:= 1200);
END_VAR
mainLamp(input:=S4_1d, output => S12_1);
END_FUNCTION_BLOCK

(* POU Global/LockMode, ST *)
FUNCTION_BLOCK LockMode
VAR_INPUT
END_VAR
VAR_OUTPUT
END_VAR
VAR
	Button: Button;
	allShaders: ARRAY [0..6] OF POINTER TO Shader;
	i: INT;
END_VAR
button(input:=H9_2c AND H9_2d);

allShaders[0]:= ADR(shader_kuchnia);
allShaders[1]:= ADR(shader_taras);
allShaders[2]:= ADR(shader_kominek);
allShaders[3]:= ADR(shader_gabinet);
allShaders[4]:= ADR(shader_lazienka);
allShaders[5]:= ADR(shader_sypialnia); (* close only *)
allShaders[6]:= ADR(shader_kotlownia); (* close only *)

IF button.longPressed THEN
	FOR i := 0 TO 6 DO
		allShaders[i]^.closeImpulse := 1;
	END_FOR
END_IF

IF button.fallingEdge THEN
	FOR i := 0 TO 4 DO
		allShaders[i]^.openImpulse := 1;
	END_FOR
END_IF
END_FUNCTION_BLOCK

(* POU V2, ST *)
PROGRAM V2
VAR
	test:INT;
	tmp:BOOL;
	block:EdgeDetection := (onRisingEdge:=1, onFallingEdge:=0);
END_VAR
block(input:=S2_2a, output=>tmp);
IF tmp THEN
	test := test + 1;
END_IF
END_PROGRAM

(* POU clock01s, ST *)
PROGRAM clock01s
VAR
END_VAR
clock01secImpulse:=1;
END_PROGRAM

(* POU Interrupt_0, ST *)
PROGRAM Interrupt_0
VAR
END_VAR
 %QX0.0 := 1;
END_PROGRAM

(* POU Configuration/MODBUS_CONFIGURATION, ST *)
PROGRAM MODBUS_CONFIGURATION
VAR                                
END_VAR                            
(*                                 
   <?xml version="1.0" encoding="UTF-16" standalone="yes"?>
<network xml_structure_version="1" xml_feature_version="1">
	<generator_settings minRTUTaskCycleTimeMs="5" minEthaskCycleTimeMs="5" ethSlaveMultiplier="0.1" rtuInterfaceMultiplier="0.1" taskGeneration="true"/>
</network>
                              
*)                                 
;                                  
END_PROGRAM
